// TIA Portal project "Paketband_mit_Hoehe_2" (V20)

(* hardware
DEVICE "S7-1500/ET200MP-Station_1"  S7-1500 station
   slot 0: "Profilschiene_0"  Rack  6ES7 590-1***0-0AA0
   slot 1: "PLC_1"  CPU 1513-1 PN  6ES7 513-1AM03-0AB0  V4.0
      slot 3: "CPU-Display_1"  6ES7591-1AA00-0AA0
      slot 32768: "PROFINET-Schnittstelle_1"  X1
         slot 32769: "Port_1"  X1 P1
         slot 32770: "Port_2"  X1 P2
      slot 34817: "Virtual CP interface port_1"  Virtual CP interface port  Virtual CP interface port FW V4.0
   slot 2: "DI 16x24VDC BA_1"  DI 16x24VDC BA  6ES7 521-1BH10-0AA0  V1.1
   slot 3: "DQ 16x24VDC/0.5A ST_1"  DQ 16x24VDC/0.5A ST  6ES7 522-1BH00-0AB0  V2.0
   slot 4: "AI 8xU/I/R/RTD BA_1"  AI 8xU/I/R/RTD BA  6ES7 531-7QF00-0AB0  V1.0
   slot 5: "AQ 8xU/I HS_1"  AQ 8xU/I HS  6ES7 532-5HF00-0AB0  V2.2
   slot 6: "AI 8xU/I/R/RTD BA_2"  AI 8xU/I/R/RTD BA  6ES7 531-7QF00-0AB0  V1.0
   slot 7: "AQ 8xU/I HS_2"  AQ 8xU/I HS  6ES7 532-5HF00-0AB0  V2.2
*)

// ===== PLC "PLC_1"  CPU 1513-1 PN =====

VAR_GLOBAL   // PLC tag table "Standard-Variablentabelle"
   "PlcLabConnectIn01" AT %ID32760 : DWord;
   "PlcLabConnectIn02" AT %ID32764 : DWord;
   "PlcLabConnectOut01" AT %QD32760 : DWord;
   "PlcLabConnectOut02" AT %QD32764 : DWord;
   "Clock_Byte" AT %MB0 : Byte;
   "Clock_10Hz" AT %M0.0 : Bool;
   "Clock_5Hz" AT %M0.1 : Bool;
   "Clock_2.5Hz" AT %M0.2 : Bool;
   "Clock_2Hz" AT %M0.3 : Bool;
   "Clock_1.25Hz" AT %M0.4 : Bool;
   "Clock_1Hz" AT %M0.5 : Bool;
   "Clock_0.625Hz" AT %M0.6 : Bool;
   "Clock_0.5Hz" AT %M0.7 : Bool;
   "Tag_1" AT %MW2 : Int;
END_VAR

VAR_GLOBAL   // PLC tag table "Ausgaenge"
   "M1" AT %Q0.0 : Bool;   // Motor Förderband
   "H1" AT %Q0.1 : Bool;   // Meldeleuchte grün (Kleines Paket)
   "H2" AT %Q0.2 : Bool;   // Meldeleuchte gelb (Mittleres Paket)
   "H3" AT %Q0.3 : Bool;   // Meldeleuchte rot (Großes Paket)
   "H4" AT %Q0.4 : Bool;   // Leuchte Starttaster
   "H5" AT %Q0.5 : Bool;   // Leuchte Stopptaster
   "D1" AT %QD30 : DInt;   // Zähler (Kleine Pakete)
   "D2" AT %QD34 : DInt;   // Zähler (Mittlere Pakete)
   "D3" AT %QD38 : DInt;   // Zähler (Große Pakete)
   "D4" AT %QD42 : DInt;   // Gesamtzähler
   "M2" AT %A1.0 : Bool;   // Sortierer
   "2M1" AT %A1.1 : Bool;   // Sortierer (Links)
   "2M2" AT %A1.2 : Bool;   // Sortierer (Rechts)
END_VAR

VAR_GLOBAL   // PLC tag table "Eingaenge"
   "S1" AT %I0.0 : Bool;   // Starttaster
   "S2" AT %I0.1 : Bool;   // Stopptaster
   "1b1" AT %I0.2 : Bool;   // Sensor (Kleine Pakete)
   "1b2" AT %I0.3 : Bool;   // Sensor (Mittlere Pakete)
   "1b3" AT %I0.4 : Bool;   // Sensor (Große Pakete)
   "2b1" AT %E0.5 : Bool;   // Lichtsensor (Links)
   "3b1" AT %E0.6 : Bool;   // Lichtsensor (Mitte)
   "4b1" AT %E0.7 : Bool;   // Lichtsensor (Rechts)
END_VAR

DATA_BLOCK "Datenbaustein_1"   // DB2
{ S7_Optimized_Access := 'TRUE' }
VERSION : 0.1
   VAR
      Betriebsart : Struct
         Anlage_aktiv : Bool;
      END_STRUCT;
      Bauteilhoehe : Struct
         Klein : Bool;
         Mittel : Bool;
         Groß : Bool;
      END_STRUCT;
   END_VAR
   VAR RETAIN
      Betriebsdaten : Struct
         Zaehler : Struct
            Klein : DInt;
            Mittel : DInt;
            Groß : DInt;
            Gesamt : DInt;
         END_STRUCT;
         Betriebsstundenzaehler : LTime;
      END_STRUCT;
   END_VAR
   VAR
      Sonstiges : Struct
         Warteliste : Array[0..10] of Int;
         I_Warteliste : Int;   // Iterator der Warteliste
         Klein_aus : Bool;   // Kleines Paket hat die Anlage verlassen
         Mittel_aus : Bool;   // Mittleres Paket hat die Anlage verlassen
         Groß_aus : Bool;   // Großes Paket hat die Anlage verlassen
         Allgemein_aus : Bool;   // Ein Paket hat die Anlage verlassen
         Klein_zaehlen : Bool;
         Mittel_zaehlen_1 : Bool;
         Mittel_zaehlen_2 : Bool;
         Groß_zaehlen : Bool;
      END_STRUCT;
   END_VAR
BEGIN
END_DATA_BLOCK

// folder: System blocks/Program resources

DATA_BLOCK "IEC_Timer_0_DB_1"   // DB1
{ S7_Optimized_Access := 'TRUE' }
AUTHOR : Simatic
FAMILY : IEC
NAME : IEC_LTMR
VERSION : 1.0
// stored: InstanceOfName IEC_LTIMER
"IEC_LTIMER"
BEGIN
END_DATA_BLOCK

// folder: (top level)

FUNCTION "Bandsteuerung" : Void   // FC1, FBD
{ S7_Optimized_Access := 'TRUE' }
VERSION : 0.1
   VAR_TEMP   // added for the SCL form of the ladder/FBD networks
      _w1 : Bool;
      _w2 : Bool;
   END_VAR
BEGIN

REGION Network 1: Förderbandsteuerung
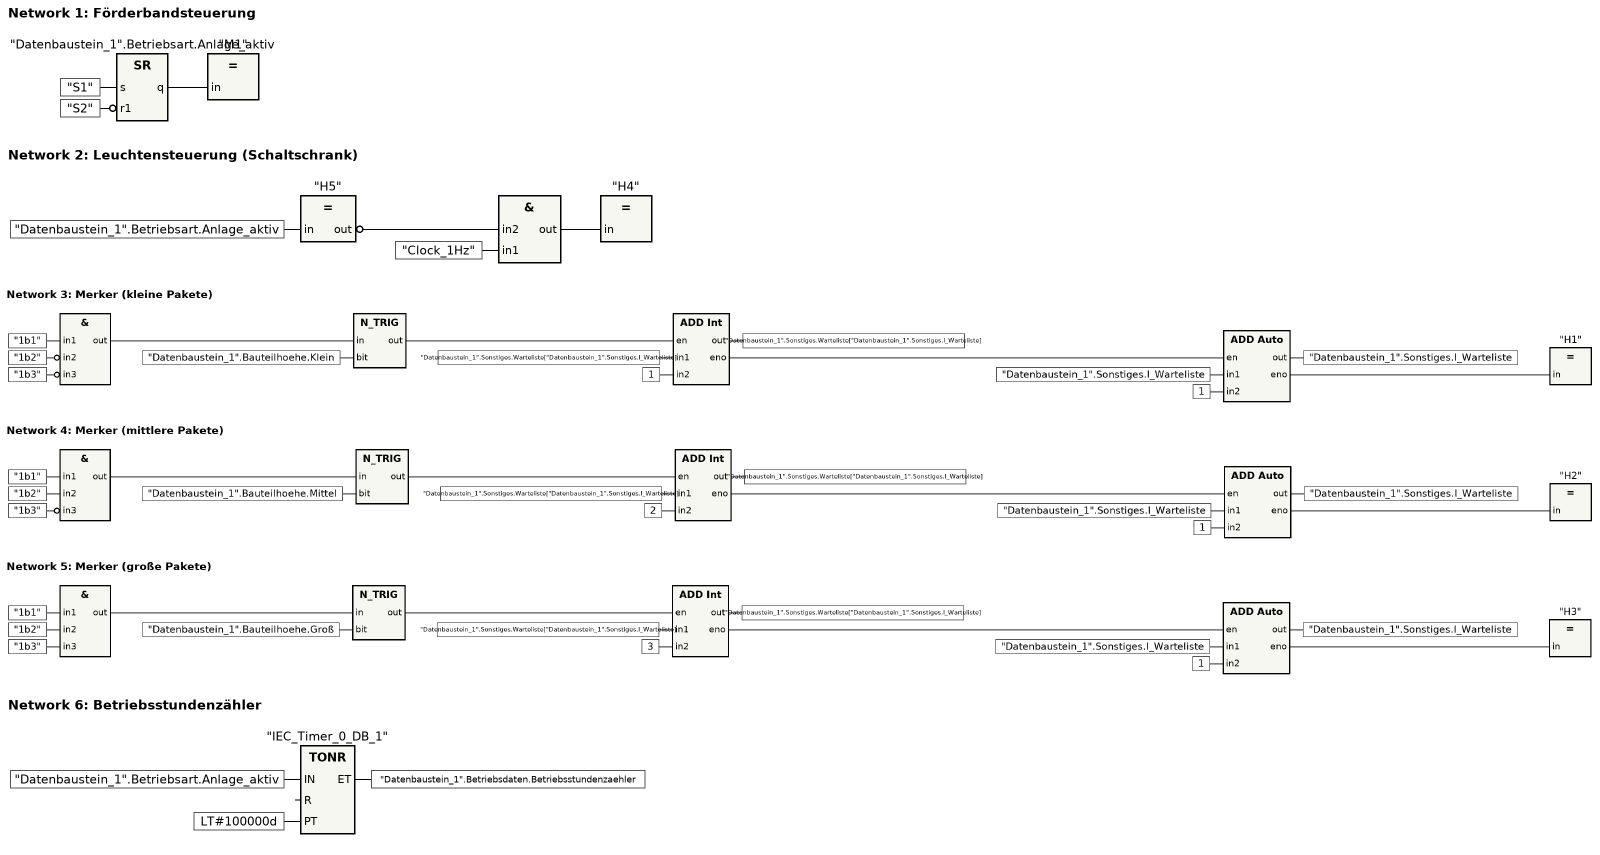
   IF "S1" THEN
       "Datenbaustein_1".Betriebsart.Anlage_aktiv := TRUE;   // SR flip-flop
   END_IF;
   IF NOT "S2" THEN "Datenbaustein_1".Betriebsart.Anlage_aktiv := FALSE; END_IF;
   "M1" := "Datenbaustein_1".Betriebsart.Anlage_aktiv;
END_REGION

REGION Network 2: Leuchtensteuerung (Schaltschrank)
   "H5" := "Datenbaustein_1".Betriebsart.Anlage_aktiv;
   "H4" := NOT "Datenbaustein_1".Betriebsart.Anlage_aktiv AND "Clock_1Hz";
END_REGION

REGION Network 3: Merker (kleine Pakete)
   #_w1 := "1b1" AND NOT "1b2" AND NOT "1b3";
   #_w2 := NOT #_w1 AND "Datenbaustein_1".Bauteilhoehe.Klein;   // falling edge
   "Datenbaustein_1".Bauteilhoehe.Klein := #_w1;
   IF #_w2 THEN
       "Datenbaustein_1".Sonstiges.Warteliste["Datenbaustein_1".Sonstiges.I_Warteliste] := "Datenbaustein_1".Sonstiges.Warteliste["Datenbaustein_1".Sonstiges.I_Warteliste] + 1;
       "Datenbaustein_1".Sonstiges.I_Warteliste := "Datenbaustein_1".Sonstiges.I_Warteliste + 1;
   END_IF;
   "H1" := #_w2;
END_REGION

REGION Network 4: Merker (mittlere Pakete)
   #_w1 := "1b1" AND "1b2" AND NOT "1b3";
   #_w2 := NOT #_w1 AND "Datenbaustein_1".Bauteilhoehe.Mittel;   // falling edge
   "Datenbaustein_1".Bauteilhoehe.Mittel := #_w1;
   IF #_w2 THEN
       "Datenbaustein_1".Sonstiges.Warteliste["Datenbaustein_1".Sonstiges.I_Warteliste] := "Datenbaustein_1".Sonstiges.Warteliste["Datenbaustein_1".Sonstiges.I_Warteliste] + 2;
       "Datenbaustein_1".Sonstiges.I_Warteliste := "Datenbaustein_1".Sonstiges.I_Warteliste + 1;
   END_IF;
   "H2" := #_w2;
END_REGION

REGION Network 5: Merker (große Pakete)
   #_w1 := "1b1" AND "1b2" AND "1b3";
   #_w2 := NOT #_w1 AND "Datenbaustein_1".Bauteilhoehe.Groß;   // falling edge
   "Datenbaustein_1".Bauteilhoehe.Groß := #_w1;
   IF #_w2 THEN
       "Datenbaustein_1".Sonstiges.Warteliste["Datenbaustein_1".Sonstiges.I_Warteliste] := "Datenbaustein_1".Sonstiges.Warteliste["Datenbaustein_1".Sonstiges.I_Warteliste] + 3;
       "Datenbaustein_1".Sonstiges.I_Warteliste := "Datenbaustein_1".Sonstiges.I_Warteliste + 1;
   END_IF;
   "H3" := #_w2;
END_REGION

REGION Network 6: Betriebsstundenzähler
   "IEC_Timer_0_DB_1".TONR(IN := "Datenbaustein_1".Betriebsart.Anlage_aktiv,
                           PT := LT#100000d,
                           ET => "Datenbaustein_1".Betriebsdaten.Betriebsstundenzaehler);
END_REGION
END_FUNCTION

FUNCTION "Sortiersteuerung" : Void   // FC2, FBD
{ S7_Optimized_Access := 'TRUE' }
VERSION : 0.1
   VAR_TEMP   // added for the SCL form of the ladder/FBD networks
      _w1 : Bool;
      _w2 : Bool;
   END_VAR
BEGIN

REGION Network 1: Sortierer
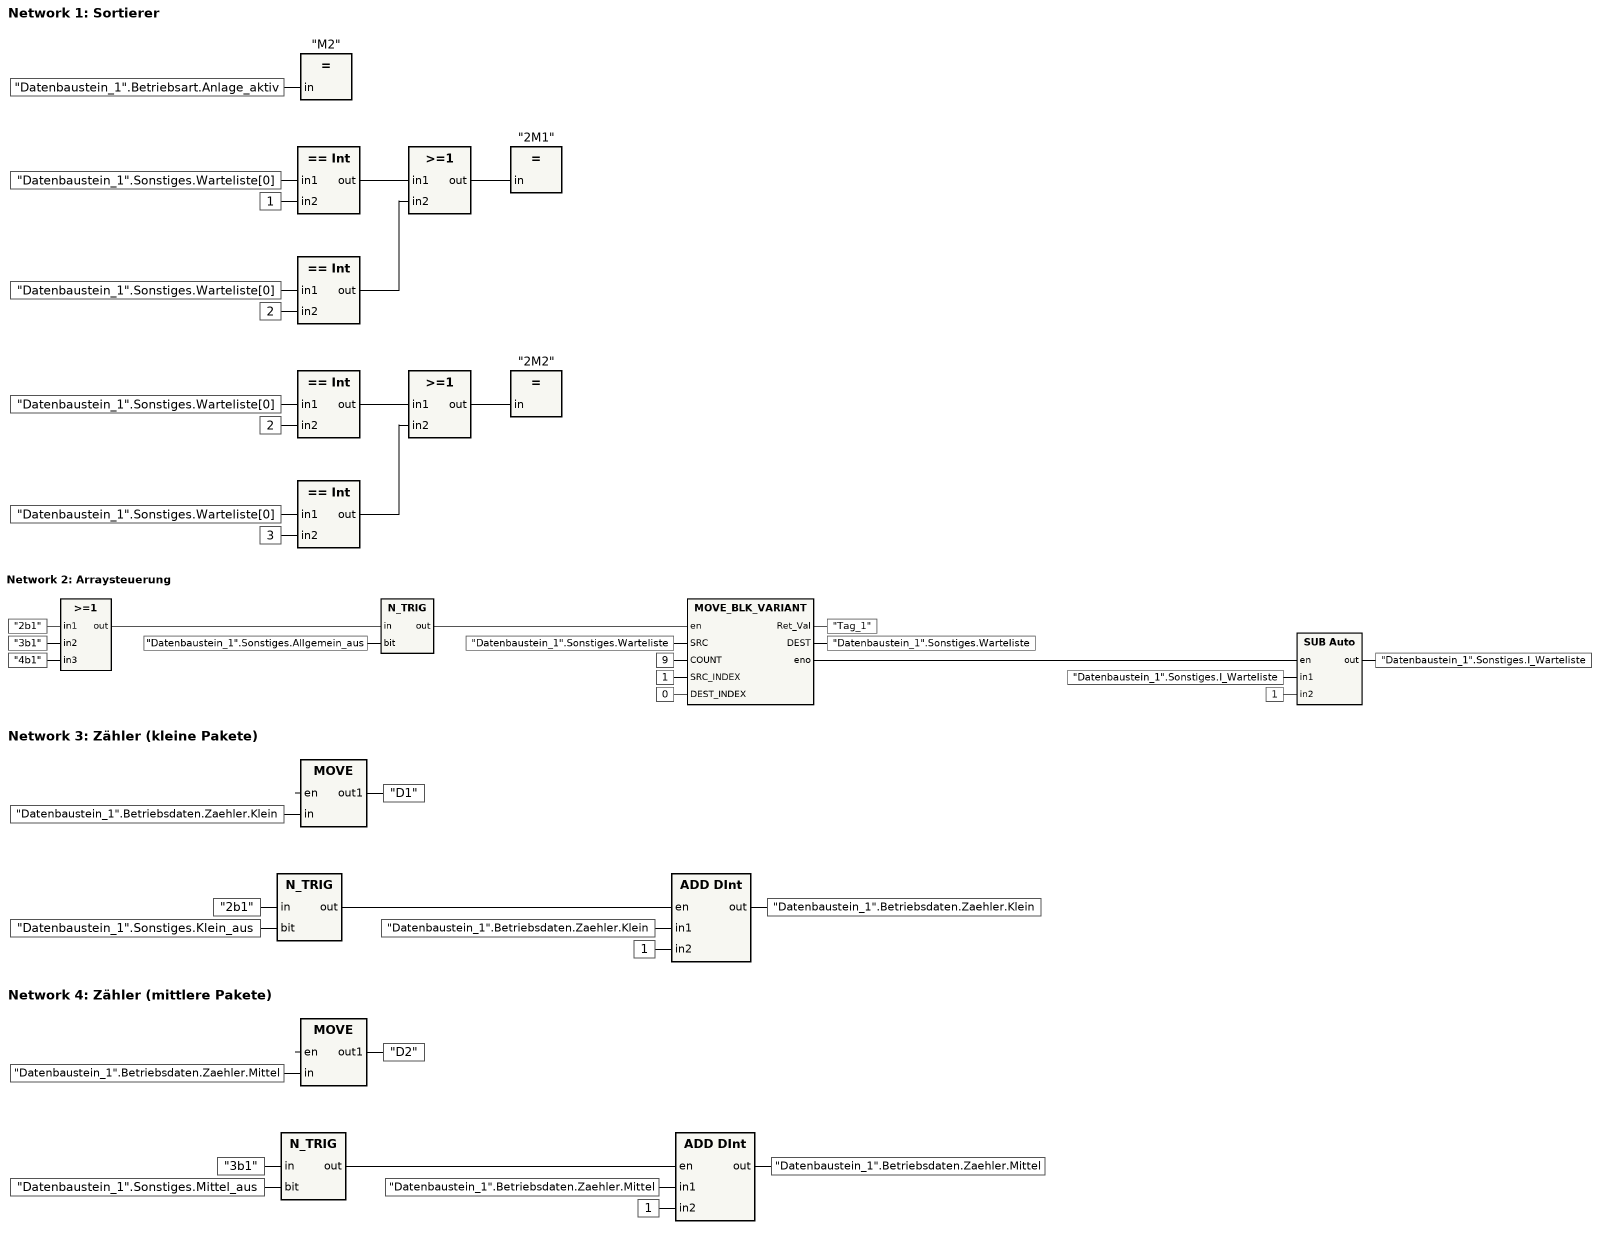
   "M2" := "Datenbaustein_1".Betriebsart.Anlage_aktiv;
   "2M1" := ("Datenbaustein_1".Sonstiges.Warteliste[0] = 1) OR ("Datenbaustein_1".Sonstiges.Warteliste[0] = 2);
   "2M2" := ("Datenbaustein_1".Sonstiges.Warteliste[0] = 2) OR ("Datenbaustein_1".Sonstiges.Warteliste[0] = 3);
END_REGION

REGION Network 2: Arraysteuerung
   // ENO of a box is taken as its EN; it also drops when the box reports an error
   #_w1 := "2b1" OR "3b1" OR "4b1";
   #_w2 := NOT #_w1 AND "Datenbaustein_1".Sonstiges.Allgemein_aus;   // falling edge
   "Datenbaustein_1".Sonstiges.Allgemein_aus := #_w1;
   IF #_w2 THEN
       "Tag_1" := MOVE_BLK_VARIANT(SRC := "Datenbaustein_1".Sonstiges.Warteliste,
                               COUNT := 9,
                               SRC_INDEX := 1,
                               DEST_INDEX := 0,
                               DEST => "Datenbaustein_1".Sonstiges.Warteliste);
       "Datenbaustein_1".Sonstiges.I_Warteliste := "Datenbaustein_1".Sonstiges.I_Warteliste - 1;
   END_IF;
END_REGION

REGION Network 3: Zähler (kleine Pakete)
   "D1" := "Datenbaustein_1".Betriebsdaten.Zaehler.Klein;
   #_w1 := NOT "2b1" AND "Datenbaustein_1".Sonstiges.Klein_aus;   // falling edge
   "Datenbaustein_1".Sonstiges.Klein_aus := "2b1";
   IF #_w1 THEN
       "Datenbaustein_1".Betriebsdaten.Zaehler.Klein := "Datenbaustein_1".Betriebsdaten.Zaehler.Klein + 1;
   END_IF;
END_REGION

REGION Network 4: Zähler (mittlere Pakete)
   "D2" := "Datenbaustein_1".Betriebsdaten.Zaehler.Mittel;
   #_w1 := NOT "3b1" AND "Datenbaustein_1".Sonstiges.Mittel_aus;   // falling edge
   "Datenbaustein_1".Sonstiges.Mittel_aus := "3b1";
   IF #_w1 THEN
       "Datenbaustein_1".Betriebsdaten.Zaehler.Mittel := "Datenbaustein_1".Betriebsdaten.Zaehler.Mittel + 1;
   END_IF;
END_REGION

REGION Network 5: Zähler (große Pakete)
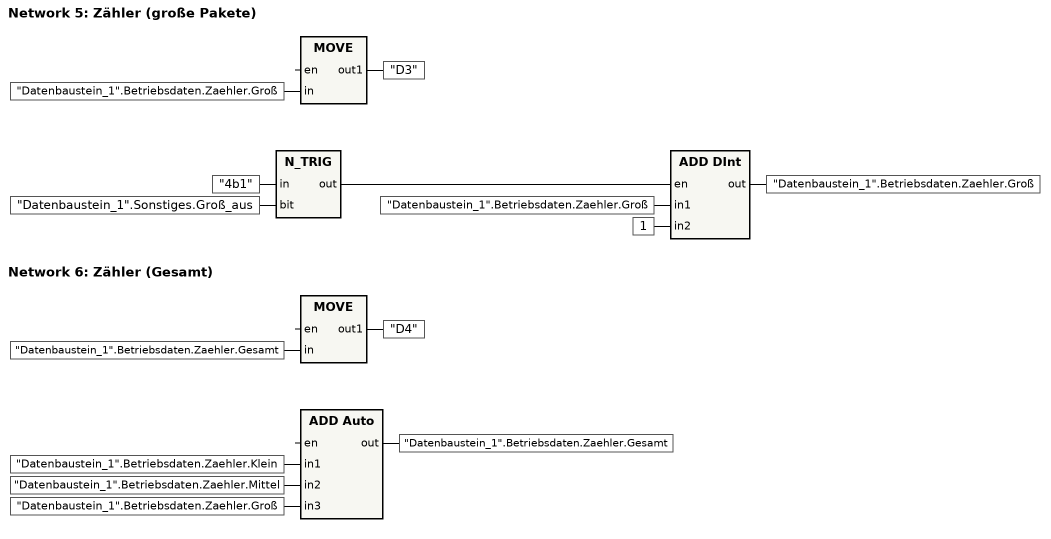
   "D3" := "Datenbaustein_1".Betriebsdaten.Zaehler.Groß;
   #_w1 := NOT "4b1" AND "Datenbaustein_1".Sonstiges.Groß_aus;   // falling edge
   "Datenbaustein_1".Sonstiges.Groß_aus := "4b1";
   IF #_w1 THEN
       "Datenbaustein_1".Betriebsdaten.Zaehler.Groß := "Datenbaustein_1".Betriebsdaten.Zaehler.Groß + 1;
   END_IF;
END_REGION

REGION Network 6: Zähler (Gesamt)
   "D4" := "Datenbaustein_1".Betriebsdaten.Zaehler.Gesamt;
   "Datenbaustein_1".Betriebsdaten.Zaehler.Gesamt := "Datenbaustein_1".Betriebsdaten.Zaehler.Klein + "Datenbaustein_1".Betriebsdaten.Zaehler.Mittel + "Datenbaustein_1".Betriebsdaten.Zaehler.Groß;
END_REGION
END_FUNCTION

ORGANIZATION_BLOCK "Main"   // OB1, FBD, ProgramCycle
TITLE = "Main Program Sweep (Cycle)"
{ S7_Optimized_Access := 'TRUE' }
VERSION : 0.1
   VAR_INPUT
      Initial_Call : Bool;   // Initial call of this OB
      Remanence : Bool;   // =True, if remanent data are available
   END_VAR
   VAR_TEMP   // added for the SCL form of the ladder/FBD networks
      _w1 : Bool;
   END_VAR
BEGIN

REGION Network 1
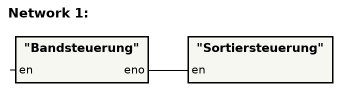
   "Bandsteuerung"(ENO => #_w1);
   IF #_w1 THEN "Sortiersteuerung"(); END_IF;
END_REGION
END_ORGANIZATION_BLOCK